Universal Robots PolyScope program: groep_pi_robot_gripper.urp

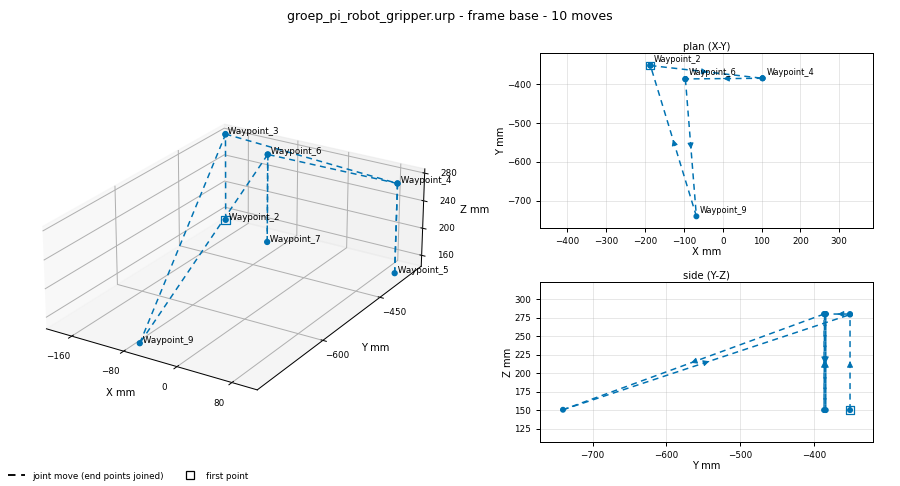
[picture p0: tool path of groep_pi_robot_gripper.urp in frame base, 10 of 10 moves have a stored position in this frame; points joined in program order, loops and branches not executed]
Program groep_pi_robot_gripper (installation=default directory=/programs/usbdisk_0 createdIn=3.15.6.106324 lastSavedIn=3.15.6.106324 robotSerialNumber=2017354085)
Calibrated DH parameters: a=[0.000173, -0.08184, -0.390569, 0.000014, 0.000061, 0]; d=[0.089465, 325.63058, -320.968373, -4.551618, 0.094907, 0.082699]; alpha=[1.570634, -0.001282, 0.007518, 1.570171, -1.57068, 0]; deltaTheta=[0.000011, -1.377212, 1.46664, -0.089508, -0.000013, 0.000027]
Robot Program (runOnlyOnce=false)
  Folder Object_1
    MoveJ speed 60 deg/s, acceleration 80 deg/s^2 (useActiveTCP=true)
      Waypoint Waypoint_2: TCP in base x=-186.232 y=-351.629 z=150.014 mm, rx=-0.3692 ry=-3.0779 rz=-0.0129 rad; joints [-101.309, -91.819, -134.143, -44.341, 87.851, 2.632] deg
    Wait DigitalInput pin=digital_in[6]; digitalValue=1
    MoveJ speed 60 deg/s, acceleration 80 deg/s^2 (useActiveTCP=true)
      Waypoint Waypoint_3: TCP in base x=-186.22 y=-351.64 z=279.949 mm, rx=-0.3693 ry=-3.078 rz=-0.0129 rad; joints [-101.265, -79.431, -122.293, -68.573, 87.95, 2.535] deg
      Waypoint Waypoint_4: TCP in base x=102.584 y=-384.454 z=279.99 mm, rx=0.7803 ry=-3.0004 rz=0.0115 rad; joints [-58.424, -79.429, -122.289, -68.576, 87.965, 2.538] deg
      Waypoint Waypoint_5: TCP in base x=102.538 y=-384.462 z=149.975 mm, rx=0.7802 ry=-3.0004 rz=0.0114 rad; joints [-58.473, -91.825, -134.145, -44.33, 87.871, 2.636] deg
        Until REACHED_WAYPOINT (allowActions=true)
          Set SingleDigitalPulseActionState SingleDigitalPulseActionState(hiPulseInSeconds=0.01, pin=digital_out[6])
          Wait Sleep waitTime=0.5
  Folder Object_2
    Wait DigitalInput pin=digital_in[6]; digitalValue=1
    MoveJ speed 60 deg/s, acceleration 80 deg/s^2 (useActiveTCP=true)
      Waypoint Waypoint_4: TCP in base x=102.584 y=-384.454 z=279.99 mm, rx=0.7803 ry=-3.0004 rz=0.0115 rad; joints [-58.424, -79.429, -122.289, -68.576, 87.965, 2.538] deg
      Waypoint Waypoint_6: TCP in base x=-96.13 y=-386.128 z=279.905 mm, rx=0.0063 ry=-3.0997 rz=-0.0053 rad; joints [-87.345, -79.437, -122.292, -68.578, 87.965, 2.54] deg
      Waypoint Waypoint_7: TCP in base x=-96.134 y=-386.732 z=150.016 mm, rx=0.0063 ry=-3.0995 rz=-0.0109 rad; joints [-87.391, -91.894, -133.988, -44.638, 87.874, 2.64] deg
        Until REACHED_WAYPOINT (allowActions=true)
          Set SingleDigitalPulseActionState SingleDigitalPulseActionState(hiPulseInSeconds=0.01, pin=digital_out[6])
          Wait Sleep waitTime=0.5
      Wait DigitalInput pin=digital_in[6]; digitalValue=1
      Waypoint Waypoint_8: TCP in base x=-96.117 y=-386.757 z=280 mm, rx=0.0065 ry=-3.0994 rz=-0.0109 rad; joints [-87.346, -79.55, -122.135, -68.833, 87.963, 2.534] deg
      Waypoint Waypoint_9: TCP in base x=-67.844 y=-740.024 z=150.471 mm, rx=0.0307 ry=-3.101 rz=0.0495 rad; joints [-86.386, -132.188, -74.314, -61.798, 87.954, 2.536] deg
        Until REACHED_WAYPOINT (allowActions=true)
          Set SingleDigitalPulseActionState SingleDigitalPulseActionState(hiPulseInSeconds=0.01, pin=digital_out[6])
          Wait Sleep waitTime=0.5
      Wait DigitalInput pin=digital_in[6]; digitalValue=1
      Waypoint Waypoint_1: TCP in base x=-186.261 y=-351.668 z=279.217 mm, rx=-0.3691 ry=-3.0779 rz=-0.0129 rad; joints [-101.27, -79.48, -122.369, -68.448, 87.943, 2.527] deg
      Set SingleDigitalPulseActionState SingleDigitalPulseActionState(hiPulseInSeconds=0.1, pin=digital_out[5])
      Halt
